(* CODESYS project %VISU%Visualization.xml

Project tree, tasks and I/O mapping:
  visualisation Visualization
*)

// /Visualization
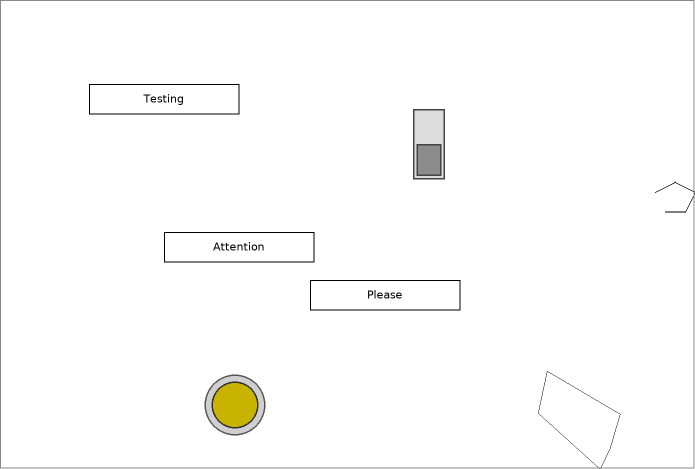
VISUALIZATION Visualization  // 695x469
    Rectangle (89,84 150x30), "Testing"
    RoundedRectangle (164,232 150x30), "Attention"
    Polyline (655,192) (675,182) (695,192) (685,212) (665,212)
    Polygon (538,413) (547,371) (620,414) (610,448) (600,469)
    DipSwitch (394,109 70x70), behaviour: TOGGLE, style: Switch-DipSwitch-Gray
    Lamp1 (200,370 70x70), style: Lamp-Lamp1-Yellow
    RoundedRectangle (310,280 150x30), "Please"
END_VISUALIZATION
